FUNCTION_BLOCK ReleaseHybrid EXTENDS ReleaseClient
VAR_INPUT
	bReleaseAckIn : BOOL;
END_VAR

VAR_OUTPUT
	bSetRelease : BOOL;
	bLastHandshakeSuccesfulHybrid : BOOL;
END_VAR


VAR
	fbReleaseAckInEvent : R_TRIG;
	fbSetReleaseEvent : R_TRIG;
	fbHandshakeSuccessfulEvent : R_TRIG;
END_VAR

SUPER^();
fbReleaseAckInEvent(CLK:=bReleaseAckIn);
fbSetReleaseEvent(CLK:=bSetRelease);

IF fbReleaseAckInEvent.Q
THEN
	OnReleaseAckIn();
END_IF

IF fbSetReleaseEvent.Q
THEN
	OnSetRelease();
END_IF

IF fbHandshakeSuccessfulEvent.Q
THEN	
	bLastHandshakeSuccesful := TRUE;
END_IF

METHOD OnHandshakeSuccessful : BOOL
VAR_INPUT
END_VAR
END_METHOD

METHOD OnReleaseAckIn : BOOL
VAR_INPUT
END_VAR
bSetRelease := FALSE;
END_METHOD

METHOD OnSetRelease : BOOL
VAR_INPUT
END_VAR
bLastHandshakeSuccesfulHybrid := FALSE;
END_METHOD

METHOD SetReleaseClient : BOOL
VAR_IN_OUT
	fbReleaseClient : ReleaseClient;
END_VAR
bReleaseAckIn := fbReleaseClient.bReleaseAckOut;
fbReleaseClient.bReleasePresent := bSetRelease;

fbHandshakeSuccessfulEvent(CLK:=fbReleaseClient.bLastHandshakeSuccesful);
END_METHOD

END_FUNCTION_BLOCK

(* stored: Version 1.1.0.1, ProductVersion 3.1.4024.2
   POU ReleaseHybrid: Id {62898187-7173-4114-9b9e-eba6cc928c84}, SpecialFunc None
   Method OnHandshakeSuccessful: Id {fd2496f1-8f28-4daf-a0ff-c614084e1ab2}
   Method OnReleaseAckIn: Id {bb7d6fda-b411-4a9f-9372-3c3c6858cebf}
   Method OnSetRelease: Id {a962a124-aa8b-4ae0-be8d-d442d919b401}
   Method SetReleaseClient: Id {412d4f81-e219-4209-895c-285c49672eb8} *)
